      NOP   0; // Hold comments
      A     #s_Mode_Manual;
      =     #o_Manual_Selected;

      A     #s_ST_Infeed1_Pos;
      =     #o_ST_Pos_Infeed1;

      A     #s_ST_Infeed2_Pos;
      =     #o_ST_Pos_Infeed2;

      A     #s_ST_Outfeed_Pos;
      =     #o_ST_Pos_Outfeed;

      A     #s_ST_Maint_Up_Pos;
      =     #o_ST_Pos_Maint_Up;

      A     #s_ST_Maint_Down_Pos;
      =     #o_ST_Pos_Maint_Down;

      A     #s_MS_Not_Auto;
      =     #o_ST_MS_Not_Automatic;

      A     #s_LCC_MS_Not_Auto;
      =     #o_ST_KS_LCC_Not_Auto;

      A     #s_ST_FieldB_NotPrsnt;
      =     #o_ST_FieldB_NotPrsnt;

      A     #s_ST_FieldB_Error;
      =     #o_ST_FieldB_Error;

      A     #s_ST_FieldB2_NotPrsnt;
      =     #o_ST_FieldB2_NotPrsnt;

      A     #s_ST_FieldB2_Error;
      =     #o_ST_FieldB2_Error;


      A     #s_ST_FieldB3_NotPrsnt;
      =     #o_ST_FieldB3_NotPrsnt;

      A     #s_ST_FieldB3_Error;
      =     #o_ST_FieldB3_Error;


      A     #s_ST_Not_At_Infeed1;
      =     #o_ST_Not_At_Infeed1;

      A     #s_ST_Not_At_Infeed2;
      =     #o_ST_Not_At_Infeed2;

      A     #s_TH_Main_Power;
      =     #o_ST_TH_Main_Power;

      A     #s_TH_Hoist_Carrier_Power;
      =     #o_TH_Hoist_Carrier_Power;

      A     #s_ST_Inf1_Gap_Not_Clr;
      =     #o_ST_Infeed1_Gap_Not_Clr;

      A     #s_ST_Inf2_Gap_Not_Clr;
      =     #o_ST_Infeed2_Gap_Not_Clr;

      A     #s_ST_Outf_Gap_Not_Clr;
      =     #o_ST_Outfeed_Gap_Not_Clr;

      A     #s_TRS_PEC_EOS_Unex_Occ;
      A     #s_TRS_PEC_SOS_Unex_Occ;
      =     #o_TRS_ST_Bag_To_Long;

      A     #s_TRS_PEC_EOS_Unex_Occ;
      AN    #o_TRS_ST_Bag_To_Long;
      =     #o_TRS_ST_PEC_EOS_Un_Oc;

      A     #s_TRS_PEC_SOS_Unex_Occ;
      AN    #o_TRS_ST_Bag_To_Long;
      =     #o_TRS_ST_PEC_SOS_Un_Oc;

      A     #s_ST_Saf_fence_infeed;
      =     #o_ST_Saf_fence_infeed;

      A     #s_ST_Saf_fence_infeed2;
      =     #o_ST_Saf_fence_infeed2;

      A     #s_ST_Saf_fence_outfeed;
      =     #o_ST_Saf_fence_outfeed;

      A     #s_ST_Safety_Relais;
      =     #o_ST_Safety_Relais;

      A     #s_SWS_ST_Move_Time_Out;
      =     #o_SWS_ST_Move_Time_Out;

      AN    #s_ST_Homing_Done;
      =     #o_SWS_ST_Not_Homed;

      A     #s_SWS_ST_Running;
      =     #o_SWS_ST_Running;

      A     #s_SWS_Ready_To_Restart;
      O     #s_TRS_Ready_To_Restart;
      A     #s_Available_IO_Below;
      AN    #s_Mode_Manual;
      A     #i_CMD_Enable;
      AN    #s_Error_On_Zone_Level;
      =     #o_Ready_To_Restart;

      A     #s_SWS_ST_Running;
      AN    #s_SWS_Req_Stop;
      O     ;
      A     #o_TRS_ST_Running;
      AN    #s_TRS_Req_Stop;
      AN    #s_Bag_Unloaded;
      =     #o_Action_Active;

      A     #s_Mode_Semi_Infeed1;
      =     #o_ST_Fixed_Infeed1;

      A     #s_Mode_Semi_Infeed2;
      =     #o_ST_Fixed_Infeed2;

//PBB Status
      AN    #o_ST_Inf_ASI_NotPrsnt;
      AN    #o_ST_Inf_ASI_Error;
      AN    #i_PBB_Inf_Auto;
      =     #o_ST_PBB_Inf_not_Auto;

      AN    #o_ST_Inf2_ASI_NotPrsnt;
      AN    #o_ST_Inf2_ASI_Error;
      AN    #i_PBB_Inf2_Auto;
      =     #o_ST_PBB_Inf2_not_Auto;

      AN    #o_ST_Outf_ASI_NotPrsnt;
      AN    #o_ST_Outf_ASI_Error;
      AN    #i_PBB_Outf_Auto;
      =     #o_ST_PBB_Outf_not_Auto;

      A     #t_ASI_Gateway_CH_OK;
      =     #o_ASI_Gateway_CH_OK;
END_FUNCTION_BLOCK

